(* Valve Control *)

FUNCTION_BLOCK FB_Valve
  VAR_INPUT
    Open_Cmd : BOOL;
    Close_Cmd : BOOL;
    Fault_In : BOOL;
    Reset : BOOL;
  END_VAR
  VAR_OUTPUT
    Valve_Open : BOOL;
    Valve_Closed : BOOL;
    Valve_Fault : BOOL;
  END_VAR

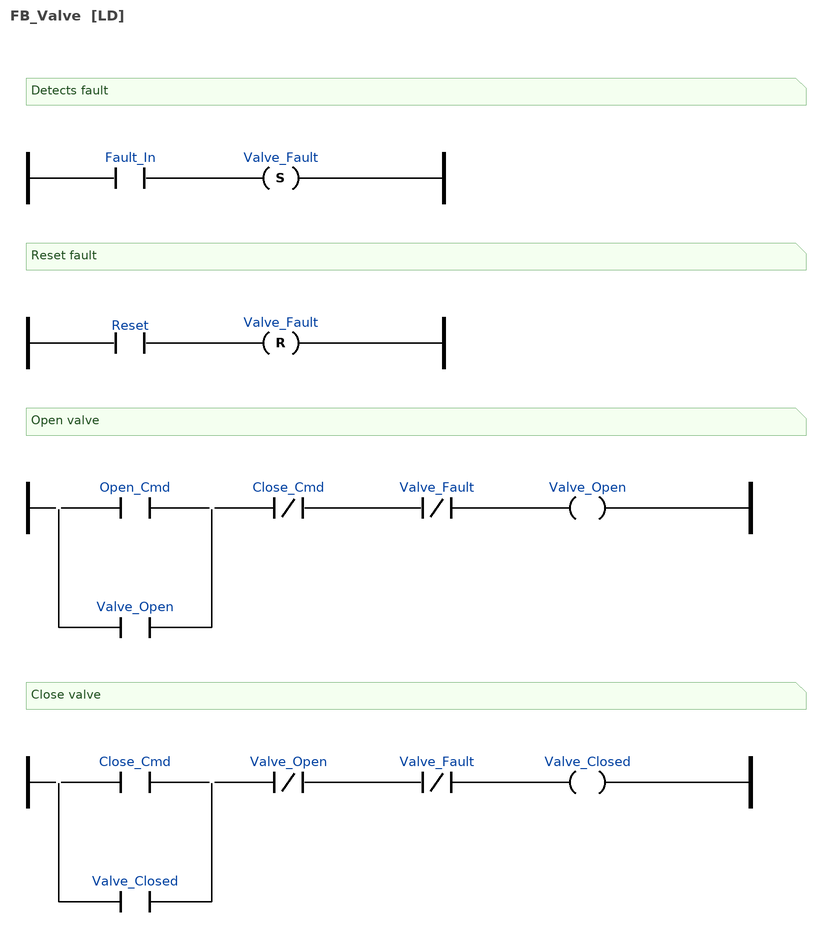
(* LD diagram, written out as Structured Text *)
(* Detects fault *)
IF Fault_In THEN Valve_Fault := TRUE; END_IF;
(* Reset fault *)
IF Reset THEN Valve_Fault := FALSE; END_IF;
(* Open valve *)
Valve_Open := (Open_Cmd OR Valve_Open) AND NOT Close_Cmd AND NOT Valve_Fault;
(* Close valve *)
Valve_Closed := (Close_Cmd OR Valve_Closed) AND NOT Valve_Open AND NOT Valve_Fault;
END_FUNCTION_BLOCK
